  - Placa_175 [part] at (1150, 250, 200) mm
  - Disco_176 [part] at (1250, 230, 200) mm
  - Placa_177 [part] at (1150, 250, 200) mm
  - Disco_178 [part] at (1250, 230, 200) mm
  - Placa_179 [part] at (1146.4, 250, 200) mm
  - Placa_180 [part] at (1150, 250, 200) mm
  - Disco_181 [part] at (1250, 230, 200) mm
  - Placa_182 [part] at (1150, 250, 200) mm
  - Placa_183 [part] at (1150, 250, 200) mm
  - Placa_184 [part] at (1150, 250, 200) mm
  - Disco_185 [part] at (1250, 230, 200) mm
  - Placa_186 [part] at (1150, 250, 200) mm
  - Disco_187 [part] at (1250, 230, 200) mm
  - Disco_188 [part] at (1250, 230, 200) mm
  - Placa_189 [part] at (1150, 250, 200) mm
  - Placa_190 [part] at (1150, 250, 200) mm
  - Placa_191 [part] at (1150, 250, 200) mm
  - Placa_192 [part] at (1150, 250, 200) mm
  - Disco_193 [part] at (1250, 230, 200) mm
  - Placa_194 [part] at (1150, 250, 200) mm
  - Placa_195 [part] at (1150, 250, 200) mm
  - Disco_196 [part] at (1250, 230, 200) mm
  - Disco_197 [part] at (1250, 230, 200) mm
  - Placa_198 [part] at (1150, 250, 200) mm
  - Disco_199 [part] at (1250, 230, 200) mm
  - Disco_200 [part] at (1250, 230, 200) mm
  - Disco_201 [part] at (1250, 230, 200) mm
  - Placa_202 [part] at (1150, 250, 200) mm
  - Placa_203 [part] at (1146.4, 250, 200) mm
  - Disco_204 [part] at (1250, 230, 200) mm
  - Placa_205 [part] at (1150, 250, 200) mm
  - Disco_206 [part] at (1250, 230, 200) mm
  - Placa_207 [part] at (1150, 250, 200) mm
  - Placa_208 [part] at (1150, 250, 200) mm
  - Disco_209 [part] at (1250, 230, 200) mm
  - Disco_210 [part] at (1250, 230, 200) mm
  - Disco_211 [part] at (1246.4, 230, 200) mm
  - Placa_212 [part] at (1150, 250, 200) mm
  - Disco_213 [part] at (1250, 230, 200) mm
  - Placa_214 [part] at (1150, 250, 200) mm
  - Placa_215 [part] at (1150, 250, 200) mm
  - Placa_216 [part] at (1150, 250, 200) mm
  - Disco_217 [part] at (1250, 230, 200) mm
  - Placa_218 [part] at (1150, 250, 200) mm
  - Disco_219 [part] at (1250, 230, 200) mm
  - Disco_220 [part] at (1246.4, 230, 200) mm
  - Disco_221 [part] at (1250, 230, 200) mm
  - Disco_222 [part] at (1250, 230, 200) mm
  - Disco_223 [part] at (1250, 230, 200) mm
  - Disco_224 [part] at (1250, 230, 200) mm
  - Disco_225 [part] at (1250, 230, 200) mm
  - Placa_226 [part] at (1150, 250, 200) mm
  - Placa_227 [part] at (1150, 250, 200) mm
  - Disco_228 [part] at (1250, 230, 200) mm
  - Disco_229 [part] at (1250, 230, 200) mm
  - Placa_230 [part] at (1150, 250, 200) mm
  - Disco_231 [part] at (1250, 230, 200) mm
  - Placa_232 [part] at (1150, 250, 200) mm
  - Placa_233 [part] at (1150, 250, 200) mm
  - Placa_234 [part] at (1150, 250, 200) mm
  - Placa_235 [part] at (1150, 250, 200) mm
  - Disco_236 [part] at (1250, 230, 200) mm
  - Disco_237 [part] at (1250, 230, 200) mm
  - Placa_238 [part] at (1150, 250, 200) mm
  - Disco_239 [part] at (1250, 230, 200) mm
  - Disco_240 [part] at (1250, 230, 200) mm
  - Placa_241 [part] at (1150, 250, 200) mm
  - Placa_242 [part] at (1150, 250, 200) mm
  - Placa_243 [part] at (1150, 250, 200) mm
  - Disco_244 [part] at (1250, 230, 200) mm
  - Disco_245 [part] at (1246.4, 230, 200) mm
  - Disco_246 [part] at (1250, 230, 200) mm
  - Placa_247 [part] at (1150, 250, 200) mm
  - Disco_248 [part] at (1250, 230, 200) mm
  - Placa_249 [part] at (1150, 250, 200) mm
  - Placa_250 [part] at (1150, 250, 200) mm
  - Disco_251 [part] at (1250, 230, 200) mm
  - Placa_252 [part] at (1150, 250, 200) mm
  - Placa_253 [part] at (1146.4, 250, 200) mm
  - Placa_254 [part] at (1150, 250, 200) mm
  - Placa_255 [part] at (1150, 250, 200) mm
  - Placa_256 [part] at (1150, 250, 200) mm
  - Placa_257 [part] at (1150, 250, 200) mm
  - Disco_258 [part] at (1250, 230, 200) mm
  - Disco_259 [part] at (1250, 230, 200) mm
  - Placa_260 [part] at (1150, 250, 200) mm
  - Placa_261 [part] at (1146.4, 250, 200) mm
  - Placa_262 [part] at (1150, 250, 200) mm
  - Disco_263 [part] at (1250, 230, 200) mm
  - Placa_264 [part] at (1150, 250, 200) mm
  - Disco_265 [part] at (1250, 230, 200) mm
  - Placa_266 [part] at (1150, 250, 200) mm
  - Placa_267 [part] at (1150, 250, 200) mm
  - Disco_268 [part] at (1250, 230, 200) mm
  - Disco_269 [part] at (1250, 230, 200) mm
  - Placa_270 [part] at (1150, 250, 200) mm
  - Disco_271 [part] at (1250, 230, 200) mm
  - Disco_272 [part] at (1250, 230, 200) mm
  - Disco_273 [part] at (1250, 230, 200) mm
  - Disco_274 [part] at (1250, 230, 200) mm
  - Placa_275 [part] at (1150, 250, 200) mm
  - Placa_276 [part] at (1150, 250, 200) mm
  - Disco_277 [part] at (1250, 230, 200) mm
  - Placa_278 [part] at (1150, 250, 200) mm
  - Disco_279 [part] at (1250, 230, 200) mm
  - Disco_280 [part] at (1250, 230, 200) mm
  - Placa_281 [part] at (1150, 250, 200) mm
  - Disco_282 [part] at (1250, 230, 200) mm
  - Disco_283 [part] at (1250, 230, 200) mm
  - Disco_284 [part] at (1250, 230, 200) mm
  - Placa_285 [part] at (1146.4, 250, 200) mm
  - Disco_286 [part] at (1250, 230, 200) mm
  - Disco_287 [part] at (1250, 230, 200) mm
  - Disco_288 [part] at (1250, 230, 200) mm
  - Disco_289 [part] at (1250, 230, 200) mm
  - Placa_290 [part] at (1150, 250, 200) mm
  - Placa_291 [part] at (1150, 250, 200) mm
  - Placa_292 [part] at (1150, 250, 200) mm
  - Disco_293 [part] at (1246.4, 230, 200) mm
  - Placa_294 [part] at (1150, 250, 200) mm
  - Disco_295 [part] at (1250, 230, 200) mm
  - Disco_296 [part] at (1250, 230, 200) mm
  - Disco_297 [part] at (1250, 230, 200) mm
  - Disco_298 [part] at (1250, 230, 200) mm
  - Disco_299 [part] at (1250, 230, 200) mm
  - Disco_300 [part] at (1250, 230, 200) mm
  - Disco_301 [part] at (1250, 230, 200) mm
  - Disco_302 [part] at (1250, 230, 200) mm
  - Disco_303 [part] at (1250, 230, 200) mm
  - Disco_304 [part] at (1250, 230, 200) mm
  - Placa_305 [part] at (1150, 250, 200) mm
  - Placa_306 [part] at (1150, 250, 200) mm
  - Placa_307 [part] at (1150, 250, 200) mm
  - Disco_308 [part] at (1250, 230, 200) mm
  - Disco_309 [part] at (1246.4, 230, 200) mm
  - Disco_310 [part] at (1250, 230, 200) mm
  - Disco_311 [part] at (1250, 230, 200) mm
  - Placa_312 [part] at (1150, 250, 200) mm
  - Disco_313 [part] at (1250, 230, 200) mm
  - Disco_314 [part] at (1250, 230, 200) mm
  - Placa_315 [part] at (1150, 250, 200) mm
  - Placa_316 [part] at (1150, 250, 200) mm
  - Disco_317 [part] at (1250, 230, 200) mm
  - Disco_338 [part] at (1246.4, 230, 200) mm
  - Disco_355 [part] at (1250, 230, 200) mm
  - Placa_356 [part] at (1150, 250, 200) mm
  - Disco_357 [part] at (1250, 230, 200) mm
  - Disco_358 [part] at (1250, 230, 200) mm
  - Disco_359 [part] at (1250, 230, 200) mm
  - Disco_360 [part] at (1250, 230, 200) mm
  - Placa_361 [part] at (1150, 250, 200) mm
  - Disco_362 [part] at (1250, 230, 200) mm
  - Placa_363 [part] at (1150, 250, 200) mm
  - Disco_364 [part] at (1246.4, 230, 200) mm
  - Placa_365 [part] at (1150, 250, 200) mm
  - Disco_366 [part] at (1250, 230, 200) mm
  - Placa_367 [part] at (1150, 250, 200) mm
  - Placa_368 [part] at (1150, 250, 200) mm
  - Disco_369 [part] at (1250, 230, 200) mm
  - Disco_370 [part] at (1250, 230, 200) mm
  - Disco_371 [part] at (1250, 230, 200) mm
  - Placa_372 [part] at (1146.4, 250, 200) mm
  - Disco_373 [part] at (1250, 230, 200) mm
  - Disco_374 [part] at (1250, 230, 200) mm
  - Disco_375 [part] at (1250, 230, 200) mm
  - Disco_376 [part] at (1250, 230, 200) mm
  - Disco_377 [part] at (1250, 230, 200) mm
  - Disco_378 [part] at (1250, 230, 200) mm
  - Placa_379 [part] at (1150, 250, 200) mm
  - Placa_380 [part] at (1146.4, 250, 200) mm
  - Placa_381 [part] at (1150, 250, 200) mm
  - Placa_382 [part] at (1150, 250, 200) mm
  - Disco_383 [part] at (1250, 230, 200) mm
  - Placa_384 [part] at (1150, 250, 200) mm
  - Placa_385 [part] at (1150, 250, 200) mm
  - Placa_386 [part] at (1150, 250, 200) mm
  - Placa_387 [part] at (1150, 250, 200) mm
  - Placa_388 [part] at (1150, 250, 200) mm
  - Placa_389 [part] at (1150, 250, 200) mm
  - Disco_390 [part] at (1250, 230, 200) mm
  - Disco_391 [part] at (1250, 230, 200) mm
  - Placa_392 [part] at (1150, 250, 200) mm
  - Disco_393 [part] at (1250, 230, 200) mm
  - Disco_394 [part] at (1250, 230, 200) mm
  - Disco_395 [part] at (1250, 230, 200) mm
  - Disco_396 [part] at (1246.4, 230, 200) mm
  - Disco_397 [part] at (1250, 230, 200) mm
  - Placa_398 [part] at (1150, 250, 200) mm
  - Placa_399 [part] at (1150, 250, 200) mm
  - Disco_400 [part] at (1250, 230, 200) mm
  - Disco_401 [part] at (1250, 230, 200) mm
  - Disco_402 [part] at (1250, 230, 200) mm
  - Disco_403 [part] at (1250, 230, 200) mm
  - Disco_404 [part] at (1246.4, 230, 200) mm
  - Placa_405 [part] at (1150, 250, 200) mm
  - Placa_406 [part] at (1150, 250, 200) mm
  - Disco_407 [part] at (1250, 230, 200) mm
  - Disco_408 [part] at (1250, 230, 200) mm
  - Disco_409 [part] at (1250, 230, 200) mm
  - Placa_410 [part] at (1150, 250, 200) mm
  - Disco_411 [part] at (1250, 230, 200) mm
  - Disco_412 [part] at (1246.4, 230, 200) mm
  - Placa_413 [part] at (1150, 250, 200) mm
  - Placa_414 [part] at (1150, 250, 200) mm
  - Placa_415 [part] at (1150, 250, 200) mm
  - Placa_416 [part] at (1150, 250, 200) mm
  - Placa_417 [part] at (1150, 250, 200) mm
  - Placa_418 [part] at (1150, 250, 200) mm
  - Disco_419 [part] at (1250, 230, 200) mm
  - Placa_420 [part] at (1146.4, 250, 200) mm
  - Disco_421 [part] at (1250, 230, 200) mm
  - Placa_422 [part] at (1150, 250, 200) mm
  - Disco_423 [part] at (1250, 230, 200) mm
  - Disco_424 [part] at (1250, 230, 200) mm
  - Disco_425 [part] at (1250, 230, 200) mm
  - Disco_426 [part] at (1250, 230, 200) mm
  - Placa_427 [part] at (1150, 250, 200) mm
  - Placa_428 [part] at (1146.4, 250, 200) mm
  - Disco_429 [part] at (1250, 230, 200) mm
  - Disco_430 [part] at (1250, 230, 200) mm
  - Disco_431 [part] at (1250, 230, 200) mm
  - Disco_432 [part] at (1250, 230, 200) mm
  - Disco_433 [part] at (1250, 230, 200) mm
  - Placa_434 [part] at (1150, 250, 200) mm
  - Disco_435 [part] at (1250, 230, 200) mm
  - Placa_436 [part] at (1146.4, 250, 200) mm
  - Placa_437 [part] at (1150, 250, 200) mm
  - Disco_438 [part] at (1250, 230, 200) mm
  - Disco_439 [part] at (1250, 230, 200) mm
  - Disco_440 [part] at (1250, 230, 200) mm
  - Placa_441 [part] at (1150, 250, 200) mm
  - Disco_442 [part] at (1250, 230, 200) mm
  - Placa_443 [part] at (1150, 250, 200) mm
  - Placa_444 [part] at (1146.4, 250, 200) mm
  - Placa_445 [part] at (1150, 250, 200) mm
  - Disco_446 [part] at (1250, 230, 200) mm
  - Disco_447 [part] at (1250, 230, 200) mm
  - Placa_448 [part] at (1150, 250, 200) mm
  - Placa_449 [part] at (1150, 250, 200) mm
  - Disco_450 [part] at (1250, 230, 200) mm
  - Disco_451 [part] at (1250, 230, 200) mm
  - Disco_452 [part] at (1246.4, 230, 200) mm
  - Placa_453 [part] at (1150, 250, 200) mm
  - Disco_454 [part] at (1250, 230, 200) mm
  - Placa_455 [part] at (1150, 250, 200) mm
  - Disco_456 [part] at (1250, 230, 200) mm
  - Placa_457 [part] at (1150, 250, 200) mm
  - Placa_458 [part] at (1150, 250, 200) mm
  - Placa_459 [part] at (1150, 250, 200) mm
  - Disco_460 [part] at (1246.4, 230, 200) mm
  - Placa_461 [part] at (1150, 250, 200) mm
  - Placa_462 [part] at (1150, 250, 200) mm
  - Placa_463 [part] at (1150, 250, 200) mm
  - Placa_464 [part] at (1150, 250, 200) mm
  - Disco_465 [part] at (1250, 230, 200) mm
  - Placa_466 [part] at (1150, 250, 200) mm
  - Placa_467 [part] at (1150, 250, 200) mm
  - Disco_468 [part] at (1246.4, 230, 200) mm
  - Disco_469 [part] at (1250, 230, 200) mm
  - Disco_470 [part] at (1250, 230, 200) mm
  - Disco_471 [part] at (1250, 230, 200) mm
  - Placa_472 [part] at (1150, 250, 200) mm
  - Placa_473 [part] at (1150, 250, 200) mm
  - Placa_474 [part] at (1150, 250, 200) mm
  - Disco_475 [part] at (1250, 230, 200) mm
  - Disco_476 [part] at (1250, 230, 200) mm
  - Placa_477 [part] at (1150, 250, 200) mm
  - Disco_478 [part] at (1250, 230, 200) mm
  - Disco_479 [part] at (1250, 230, 200) mm
  - Disco_480 [part] at (1250, 230, 200) mm
  - Disco_481 [part] at (1250, 230, 200) mm
  - Placa_482 [part] at (1150, 250, 200) mm
  - Placa_483 [part] at (1150, 250, 200) mm
  - Disco_484 [part] at (1246.4, 230, 200) mm
  - Placa_485 [part] at (1150, 250, 200) mm
  - Disco_486 [part] at (1250, 230, 200) mm
  - Placa_487 [part] at (1150, 250, 200) mm
  - Disco_488 [part] at (1250, 230, 200) mm
  - Disco_489 [part] at (1250, 230, 200) mm
  - Placa_490 [part] at (1150, 250, 200) mm
  - Placa_491 [part] at (1150, 250, 200) mm
  - Placa_492 [part] at (1146.4, 250, 200) mm
  - Disco_493 [part] at (1250, 230, 200) mm
  - Disco_494 [part] at (1250, 230, 200) mm
  - Disco_495 [part] at (1250, 230, 200) mm
  - Placa_496 [part] at (1150, 250, 200) mm
  - Disco_497 [part] at (1250, 230, 200) mm
  - Placa_498 [part] at (1150, 250, 200) mm
  - Placa_499 [part] at (1150, 250, 200) mm
  - Placa_500 [part] at (1150, 250, 200) mm
  - Disco_501 [part] at (1250, 230, 200) mm
  - Disco_502 [part] at (1246.4, 230, 200) mm
  - Placa_505 [part] at (1146.4, 250, 200) mm
  - Placa_506 [part] at (1146.4, 250, 200) mm
  - Disco_18 [part] at (1250, 230, 200) mm
  - Disco_19 [part] at (1250, 230, 200) mm
  - Disco_20 [part] at (1250, 230, 200) mm
  - Placa_21 [part] at (1150, 250, 200) mm
  - Disco_22 [part] at (1250, 230, 200) mm
  - Disco_23 [part] at (1250, 230, 200) mm
  - Disco_24 [part] at (1250, 230, 200) mm
  - Placa_25 [part] at (1150, 250, 200) mm
  - Placa_26 [part] at (1150, 250, 200) mm
  - Placa_27 [part] at (1150, 250, 200) mm
  - Placa_28 [part] at (1150, 250, 200) mm
  - Disco_29 [part] at (1250, 230, 200) mm
  - Placa_30 [part] at (1150, 250, 200) mm
  - Placa_31 [part] at (1146.4, 250, 200) mm
  - Disco_32 [part] at (1250, 230, 200) mm
  - Placa_33 [part] at (1150, 250, 200) mm
  - Disco_34 [part] at (1250, 230, 200) mm
  - Disco_35 [part] at (1250, 230, 200) mm
  - Placa_36 [part] at (1150, 250, 200) mm
  - Disco_37 [part] at (1250, 230, 200) mm
  - Placa_38 [part] at (1146.4, 250, 200) mm
  - Placa_39 [part] at (1150, 250, 200) mm
  - Placa_40 [part] at (1146.4, 250, 200) mm
  - Placa_41 [part] at (1150, 250, 200) mm
  - Placa_42 [part] at (1146.4, 250, 200) mm
  - Disco_43 [part] at (1250, 230, 200) mm
  - Placa_44 [part] at (1146.4, 250, 200) mm
  - Placa_45 [part] at (1150, 250, 200) mm
  - Disco_46 [part] at (1250, 230, 200) mm
  - Disco_89 [part] at (1250, 230, 200) mm
  - Disco_90 [part] at (1250, 230, 200) mm
  - Disco_91 [part] at (1250, 230, 200) mm
  - Disco_92 [part] at (1246.4, 230, 200) mm
  - Placa_93 [part] at (1150, 250, 200) mm
  - Disco_94 [part] at (1250, 230, 200) mm
  - Placa_95 [part] at (1150, 250, 200) mm
  - Placa_96 [part] at (1150, 250, 200) mm
  - Disco_97 [part] at (1250, 230, 200) mm
  - Placa_98 [part] at (1150, 250, 200) mm
  - Placa_99 [part] at (1146.4, 250, 200) mm
  - Disco_100 [part] at (1250, 230, 200) mm
  - Disco_101 [part] at (1250, 230, 200) mm
  - Placa_102 [part] at (1150, 250, 200) mm
  - Placa_103 [part] at (1150, 250, 200) mm
  - Placa_104 [part] at (1150, 250, 200) mm
  - Placa_105 [part] at (1150, 250, 200) mm
  - Placa_106 [part] at (1146.4, 250, 200) mm
  - Placa_107 [part] at (1150, 250, 200) mm
  - Placa_108 [part] at (1150, 250, 200) mm
  - Placa_109 [part] at (1150, 250, 200) mm
  - Disco_110 [part] at (1250, 230, 200) mm
  - Placa_111 [part] at (1150, 250, 200) mm
  - Disco_112 [part] at (1250, 230, 200) mm
  - Disco_113 [part] at (1250, 230, 200) mm
  - Placa_114 [part] at (1150, 250, 200) mm
  - Disco_115 [part] at (1250, 230, 200) mm
  - Placa_116 [part] at (1150, 250, 200) mm
  - Placa_117 [part] at (1150, 250, 200) mm
  - Placa_118 [part] at (1150, 250, 200) mm
  - Disco_119 [part] at (1246.4, 230, 200) mm
  - Placa_120 [part] at (1150, 250, 200) mm
  - Placa_121 [part] at (1150, 250, 200) mm
  - Placa_122 [part] at (1150, 250, 200) mm
  - Disco_123 [part] at (1250, 230, 200) mm
  - Placa_124 [part] at (1150, 250, 200) mm
  - Placa_125 [part] at (1150, 250, 200) mm
  - Disco_126 [part] at (1246.4, 230, 200) mm
  - Placa_127 [part] at (1150, 250, 200) mm
  - Disco_128 [part] at (1250, 230, 200) mm
  - Disco_129 [part] at (1250, 230, 200) mm
  - Placa_130 [part] at (1150, 250, 200) mm
  - Placa_131 [part] at (1150, 250, 200) mm
  - Placa_132 [part] at (1150, 250, 200) mm
  - Disco_133 [part] at (1246.4, 230, 200) mm
  - Disco_134 [part] at (1250, 230, 200) mm
  - Disco_135 [part] at (1250, 230, 200) mm
  - Disco_136 [part] at (1250, 230, 200) mm
  - Disco_137 [part] at (1250, 230, 200) mm
  - Placa_138 [part] at (1150, 250, 200) mm
  - Disco_139 [part] at (1250, 230, 200) mm
  - Disco_140 [part] at (1250, 230, 200) mm
  - Placa_23 [part] at (1146.4, 250, 200) mm
  - Disco_38 [part] at (1246.4, 230, 200) mm
  - Placa_39 [part] at (1146.4, 250, 200) mm
  - Placa_40 [part] at (1150, 250, 200) mm
  - Placa_41 [part] at (1150, 250, 200) mm
  - Placa_42 [part] at (1150, 250, 200) mm
  - Disco_43 [part] at (1250, 230, 200) mm
  - Disco_44 [part] at (1250, 230, 200) mm
  - Placa_45 [part] at (1150, 250, 200) mm
  - Placa_46 [part] at (1146.4, 250, 200) mm
  - Disco_47 [part] at (1250, 230, 200) mm
  - Disco_48 [part] at (1250, 230, 200) mm
  - Disco_49 [part] at (1250, 230, 200) mm
  - Disco_50 [part] at (1250, 230, 200) mm
  - Placa_51 [part] at (1150, 250, 200) mm
  - Placa_52 [part] at (1150, 250, 200) mm
  - Placa_53 [part] at (1150, 250, 200) mm
  - Disco_54 [part] at (1250, 230, 200) mm
  - Placa_55 [part] at (1150, 250, 200) mm
  - Placa_56 [part] at (1150, 250, 200) mm
  - Placa_57 [part] at (1150, 250, 200) mm
  - Disco_58 [part] at (1250, 230, 200) mm
  - Disco_59 [part] at (1250, 230, 200) mm
  - Placa_60 [part] at (1146.4, 250, 200) mm
  - Placa_61 [part] at (1150, 250, 200) mm
  - Disco_62 [part] at (1250, 230, 200) mm
  - Placa_63 [part] at (1150, 250, 200) mm
  - Placa_64 [part] at (1150, 250, 200) mm
  - Disco_65 [part] at (1250, 230, 200) mm
  - Disco_66 [part] at (1250, 230, 200) mm
  - Disco_67 [part] at (1246.4, 230, 200) mm
  - Disco_68 [part] at (1250, 230, 200) mm
  - Disco_69 [part] at (1250, 230, 200) mm
  - Placa_70 [part] at (1150, 250, 200) mm
  - Placa_71 [part] at (1150, 250, 200) mm
  - Disco_72 [part] at (1250, 230, 200) mm
  - Disco_73 [part] at (1250, 230, 200) mm
  - Disco_74 [part] at (1246.4, 230, 200) mm
  - Disco_75 [part] at (1250, 230, 200) mm
  - Disco_76 [part] at (1250, 230, 200) mm
  - Disco_77 [part] at (1250, 230, 200) mm
  - Disco_78 [part] at (1250, 230, 200) mm
  - Disco_79 [part] at (1250, 230, 200) mm
  - Disco_80 [part] at (1250, 230, 200) mm
  - Placa_81 [part] at (1146.4, 250, 200) mm
  - Disco_82 [part] at (1250, 230, 200) mm
  - Disco_83 [part] at (1250, 230, 200) mm
  - Placa_84 [part] at (1150, 250, 200) mm
  - Disco_85 [part] at (1250, 230, 200) mm
  - Placa_86 [part] at (1150, 250, 200) mm
  - Placa_87 [part] at (1150, 250, 200) mm
  - Placa_88 [part] at (1146.4, 250, 200) mm
  - Placa_89 [part] at (1150, 250, 200) mm
  - Placa_90 [part] at (1150, 250, 200) mm
  - Disco_91 [part] at (1250, 230, 200) mm
  - Placa_92 [part] at (1150, 250, 200) mm
  - Placa_93 [part] at (1150, 250, 200) mm
  - Placa_94 [part] at (1150, 250, 200) mm
  - Placa_95 [part] at (1146.4, 250, 200) mm
  - Disco_96 [part] at (1250, 230, 200) mm
  - Placa_97 [part] at (1150, 250, 200) mm
  - Placa_98 [part] at (1150, 250, 200) mm
  - Disco_99 [part] at (1250, 230, 200) mm
  - Placa_100 [part] at (1150, 250, 200) mm
  - Disco_101 [part] at (1250, 230, 200) mm
  - Placa_102 [part] at (1146.4, 250, 200) mm
  - Disco_103 [part] at (1250, 230, 200) mm
  - Disco_104 [part] at (1250, 230, 200) mm
  - Placa_105 [part] at (1150, 250, 200) mm
  - Placa_106 [part] at (1150, 250, 200) mm
  - Placa_107 [part] at (1150, 250, 200) mm
  - Placa_108 [part] at (1150, 250, 200) mm
  - Placa_109 [part] at (1146.4, 250, 200) mm
  - Disco_110 [part] at (1250, 230, 200) mm
  - Disco_111 [part] at (1250, 230, 200) mm
  - Disco_112 [part] at (1250, 230, 200) mm
  - Placa_113 [part] at (1150, 250, 200) mm
  - Disco_114 [part] at (1250, 230, 200) mm
  - Disco_115 [part] at (1250, 230, 200) mm
  - Placa_116 [part] at (1146.4, 250, 200) mm
  - Placa_117 [part] at (1150, 250, 200) mm
  - Placa_118 [part] at (1150, 250, 200) mm
  - Placa_119 [part] at (1150, 250, 200) mm
  - Disco_120 [part] at (1250, 230, 200) mm
  - Placa_121 [part] at (1150, 250, 200) mm
  - Placa_122 [part] at (1150, 250, 200) mm
  - Placa_123 [part] at (1146.4, 250, 200) mm
  - Disco_124 [part] at (1250, 230, 200) mm
  - Placa_125 [part] at (1150, 250, 200) mm
  - Placa_126 [part] at (1150, 250, 200) mm
  - Placa_127 [part] at (1150, 250, 200) mm
  - Disco_128 [part] at (1250, 230, 200) mm
  - Disco_129 [part] at (1250, 230, 200) mm
  - Disco_130 [part] at (1246.4, 230, 200) mm
  - Placa_131 [part] at (1150, 250, 200) mm
  - Placa_132 [part] at (1150, 250, 200) mm
  - Placa_133 [part] at (1150, 250, 200) mm
  - Placa_134 [part] at (1150, 250, 200) mm
  - Placa_135 [part] at (1150, 250, 200) mm
  - Placa_136 [part] at (1150, 250, 200) mm
  - Placa_137 [part] at (1146.4, 250, 200) mm
  - Placa_138 [part] at (1150, 250, 200) mm
  - Disco_139 [part] at (1250, 230, 200) mm
  - Disco_140 [part] at (1250, 230, 200) mm
  - Disco_141 [part] at (1250, 230, 200) mm
  - Placa_142 [part] at (1150, 250, 200) mm
  - Placa_143 [part] at (1150, 250, 200) mm
  - Disco_144 [part] at (1246.4, 230, 200) mm
  - Disco_145 [part] at (1250, 230, 200) mm
  - Placa_146 [part] at (1150, 250, 200) mm
  - Disco_147 [part] at (1250, 230, 200) mm
  - Disco_148 [part] at (1250, 230, 200) mm
  - Disco_149 [part] at (1250, 230, 200) mm
  - Disco_150 [part] at (1250, 230, 200) mm
  - Disco_151 [part] at (1246.4, 230, 200) mm
  - Disco_152 [part] at (1250, 230, 200) mm
  - Placa_153 [part] at (1150, 250, 200) mm
  - Disco_154 [part] at (1250, 230, 200) mm
  - Placa_155 [part] at (1150, 250, 200) mm
  - Disco_156 [part] at (1250, 230, 200) mm
  - Placa_157 [part] at (1150, 250, 200) mm
  - Placa_158 [part] at (1150, 250, 200) mm
  - Placa_159 [part] at (1150, 250, 200) mm
  - Disco_160 [part] at (1250, 230, 200) mm
  - Disco_161 [part] at (1250, 230, 200) mm
  - Disco_162 [part] at (1250, 230, 200) mm
  - Placa_163 [part] at (1150, 250, 200) mm
  - Placa_164 [part] at (1150, 250, 200) mm
  - Placa_165 [part] at (1146.4, 250, 200) mm
  - Placa_166 [part] at (1150, 250, 200) mm
  - Disco_167 [part] at (1250, 230, 200) mm
  - Placa_168 [part] at (1150, 250, 200) mm
  - Disco_169 [part] at (1250, 230, 200) mm
  - Placa_170 [part] at (1150, 250, 200) mm
  - Placa_171 [part] at (1150, 250, 200) mm
  - Placa_172 [part] at (1146.4, 250, 200) mm
  - Disco_173 [part] at (1250, 230, 200) mm
  - Disco_174 [part] at (1250, 230, 200) mm
  - Disco_175 [part] at (1250, 230, 200) mm
  - Placa_176 [part] at (1150, 250, 200) mm
  - Disco_177 [part] at (1250, 230, 200) mm
  - Placa_178 [part] at (1150, 250, 200) mm
  - Disco_179 [part] at (1246.4, 230, 200) mm
  - Placa_180 [part] at (1150, 250, 200) mm
  - Disco_181 [part] at (1250, 230, 200) mm
  - Disco_182 [part] at (1250, 230, 200) mm
  - Disco_183 [part] at (1250, 230, 200) mm
  - Placa_184 [part] at (1150, 250, 200) mm
  - Placa_185 [part] at (1150, 250, 200) mm
  - Disco_186 [part] at (1246.4, 230, 200) mm
  - Disco_187 [part] at (1250, 230, 200) mm
  - Placa_188 [part] at (1150, 250, 200) mm
  - Placa_189 [part] at (1150, 250, 200) mm
  - Disco_190 [part] at (1250, 230, 200) mm
  - Placa_191 [part] at (1150, 250, 200) mm
  - Placa_192 [part] at (1150, 250, 200) mm
  - Disco_193 [part] at (1246.4, 230, 200) mm
  - Disco_194 [part] at (1250, 230, 200) mm
  - Disco_195 [part] at (1250, 230, 200) mm
  - Disco_196 [part] at (1250, 230, 200) mm
  - Disco_197 [part] at (1250, 230, 200) mm
  - Placa_198 [part] at (1150, 250, 200) mm
  - Placa_199 [part] at (1150, 250, 200) mm
  - Placa_200 [part] at (1146.4, 250, 200) mm
  - Disco_201 [part] at (1250, 230, 200) mm
  - Disco_202 [part] at (1250, 230, 200) mm
  - Disco_203 [part] at (1250, 230, 200) mm
  - Placa_204 [part] at (1150, 250, 200) mm
  - Disco_205 [part] at (1250, 230, 200) mm
  - Disco_206 [part] at (1250, 230, 200) mm
  - Placa_207 [part] at (1146.4, 250, 200) mm
  - Disco_208 [part] at (1250, 230, 200) mm
  - Disco_209 [part] at (1250, 230, 200) mm
  - Placa_210 [part] at (1150, 250, 200) mm
  - Disco_211 [part] at (1250, 230, 200) mm
  - Disco_212 [part] at (1250, 230, 200) mm
  - Placa_213 [part] at (1150, 250, 200) mm
  - Placa_214 [part] at (1146.4, 250, 200) mm
  - Placa_215 [part] at (1150, 250, 200) mm
  - Disco_216 [part] at (1250, 230, 200) mm
  - Disco_217 [part] at (1250, 230, 200) mm
  - Placa_218 [part] at (1150, 250, 200) mm
  - Placa_219 [part] at (1150, 250, 200) mm
  - Disco_220 [part] at (1250, 230, 200) mm
  - Placa_221 [part] at (1146.4, 250, 200) mm
  - Placa_222 [part] at (1150, 250, 200) mm
  - Placa_223 [part] at (1150, 250, 200) mm
  - Placa_224 [part] at (1150, 250, 200) mm
  - Placa_225 [part] at (1150, 250, 200) mm
  - Disco_226 [part] at (1250, 230, 200) mm
  - Placa_227 [part] at (1150, 250, 200) mm
  - Disco_228 [part] at (1246.4, 230, 200) mm
  - Disco_229 [part] at (1250, 230, 200) mm
  - Disco_230 [part] at (1250, 230, 200) mm
  - Placa_231 [part] at (1150, 250, 200) mm
  - Disco_232 [part] at (1250, 230, 200) mm
  - Placa_233 [part] at (1150, 250, 200) mm
  - Disco_234 [part] at (1250, 230, 200) mm
  - Disco_235 [part] at (1246.4, 230, 200) mm
  - Placa_236 [part] at (1150, 250, 200) mm
  - Placa_237 [part] at (1150, 250, 200) mm
  - Disco_238 [part] at (1250, 230, 200) mm
  - Placa_239 [part] at (1150, 250, 200) mm
  - Placa_240 [part] at (1150, 250, 200) mm
  - Placa_241 [part] at (1150, 250, 200) mm
  - Placa_242 [part] at (1146.4, 250, 200) mm
  - Placa_243 [part] at (1150, 250, 200) mm
  - Disco_244 [part] at (1250, 230, 200) mm
  - Disco_245 [part] at (1250, 230, 200) mm
  - Disco_246 [part] at (1250, 230, 200) mm
  - Placa_247 [part] at (1150, 250, 200) mm
  - Disco_248 [part] at (1250, 230, 200) mm
  - Disco_249 [part] at (1246.4, 230, 200) mm
  - Disco_250 [part] at (1250, 230, 200) mm
  - Placa_251 [part] at (1150, 250, 200) mm
  - Placa_252 [part] at (1150, 250, 200) mm
  - Disco_253 [part] at (1250, 230, 200) mm
  - Placa_254 [part] at (1150, 250, 200) mm
  - Disco_255 [part] at (1250, 230, 200) mm
  - Placa_256 [part] at (1146.4, 250, 200) mm
  - Disco_257 [part] at (1250, 230, 200) mm
  - Disco_258 [part] at (1250, 230, 200) mm
  - Placa_259 [part] at (1150, 250, 200) mm
  - Disco_260 [part] at (1250, 230, 200) mm
  - Placa_261 [part] at (1150, 250, 200) mm
  - Disco_262 [part] at (1250, 230, 200) mm
  - Disco_263 [part] at (1246.4, 230, 200) mm
  - Disco_264 [part] at (1250, 230, 200) mm
  - Disco_265 [part] at (1250, 230, 200) mm
  - Disco_266 [part] at (1250, 230, 200) mm
  - Placa_267 [part] at (1150, 250, 200) mm
  - Placa_268 [part] at (1150, 250, 200) mm
  - Disco_269 [part] at (1250, 230, 200) mm
  - Placa_270 [part] at (1146.4, 250, 200) mm
  - Disco_271 [part] at (1250, 230, 200) mm
  - Placa_272 [part] at (1150, 250, 200) mm
  - Placa_273 [part] at (1150, 250, 200) mm
  - Disco_274 [part] at (1250, 230, 200) mm
  - Placa_275 [part] at (1150, 250, 200) mm
  - Placa_276 [part] at (1150, 250, 200) mm
  - Placa_277 [part] at (1146.4, 250, 200) mm
  - Placa_278 [part] at (1150, 250, 200) mm
  - Placa_279 [part] at (1150, 250, 200) mm
  - Disco_280 [part] at (1250, 230, 200) mm
  - Disco_281 [part] at (1250, 230, 200) mm
  - Disco_282 [part] at (1250, 230, 200) mm
  - Placa_283 [part] at (1150, 250, 200) mm
  - Placa_284 [part] at (1146.4, 250, 200) mm
  - Disco_285 [part] at (1250, 230, 200) mm
  - Disco_286 [part] at (1250, 230, 200) mm
  - Placa_287 [part] at (1150, 250, 200) mm
  - Disco_288 [part] at (1250, 230, 200) mm
  - Disco_289 [part] at (1250, 230, 200) mm
  - Placa_290 [part] at (1150, 250, 200) mm
  - Disco_291 [part] at (1246.4, 230, 200) mm
  - Placa_292 [part] at (1150, 250, 200) mm
  - Disco_293 [part] at (1250, 230, 200) mm
  - Placa_294 [part] at (1150, 250, 200) mm
  - Disco_295 [part] at (1250, 230, 200) mm
  - Disco_296 [part] at (1250, 230, 200) mm
  - Placa_297 [part] at (1150, 250, 200) mm
  - Placa_298 [part] at (1146.4, 250, 200) mm
  - Placa_299 [part] at (1150, 250, 200) mm
  - Placa_300 [part] at (1150, 250, 200) mm
  - Placa_301 [part] at (1150, 250, 200) mm
  - Disco_302 [part] at (1250, 230, 200) mm
  - Disco_303 [part] at (1250, 230, 200) mm
  - Disco_304 [part] at (1250, 230, 200) mm
  - Disco_305 [part] at (1246.4, 230, 200) mm
  - Disco_306 [part] at (1250, 230, 200) mm
  - Placa_307 [part] at (1150, 250, 200) mm
  - Placa_308 [part] at (1150, 250, 200) mm
  - Placa_309 [part] at (1150, 250, 200) mm
  - Placa_310 [part] at (1150, 250, 200) mm
  - Placa_311 [part] at (1150, 250, 200) mm
  - Placa_312 [part] at (1150, 250, 200) mm
  - Disco_313 [part] at (1250, 230, 200) mm
  - Placa_314 [part] at (1150, 250, 200) mm
  - Placa_315 [part] at (1150, 250, 200) mm
  - Disco_316 [part] at (1250, 230, 200) mm
  - Placa_317 [part] at (1150, 250, 200) mm
  - Disco_318 [part] at (1250, 230, 200) mm
  - Disco_358 [part] at (1250, 230, 200) mm
  - Placa_359 [part] at (1146.4, 250, 200) mm
  - Placa_360 [part] at (1146.4, 250, 200) mm
  - Placa_361 [part] at (1150, 250, 200) mm
  - Disco_362 [part] at (1250, 230, 200) mm
  - Placa_363 [part] at (1150, 250, 200) mm
  - Disco_364 [part] at (1250, 230, 200) mm
  - Placa_365 [part] at (1150, 250, 200) mm
  - Disco_366 [part] at (1250, 230, 200) mm
  - Placa_367 [part] at (1146.4, 250, 200) mm
  - Disco_368 [part] at (1250, 230, 200) mm
  - Disco_369 [part] at (1250, 230, 200) mm
  - Placa_370 [part] at (1150, 250, 200) mm
  - Disco_371 [part] at (1250, 230, 200) mm
  - Disco_372 [part] at (1250, 230, 200) mm
  - Disco_373 [part] at (1250, 230, 200) mm
  - Placa_374 [part] at (1146.4, 250, 200) mm
  - Disco_375 [part] at (1250, 230, 200) mm
  - Disco_376 [part] at (1250, 230, 200) mm
  - Disco_377 [part] at (1250, 230, 200) mm
  - Disco_378 [part] at (1250, 230, 200) mm
  - Placa_379 [part] at (1150, 250, 200) mm
  - Placa_380 [part] at (1150, 250, 200) mm
  - Placa_381 [part] at (1146.4, 250, 200) mm
  - Disco_382 [part] at (1250, 230, 200) mm
  - Disco_383 [part] at (1250, 230, 200) mm
  - Placa_384 [part] at (1150, 250, 200) mm
  - Placa_385 [part] at (1150, 250, 200) mm
  - Disco_386 [part] at (1250, 230, 200) mm
  - Placa_387 [part] at (1150, 250, 200) mm
  - Placa_388 [part] at (1146.4, 250, 200) mm
  - Placa_389 [part] at (1150, 250, 200) mm
  - Disco_390 [part] at (1250, 230, 200) mm
  - Disco_391 [part] at (1250, 230, 200) mm
  - Placa_392 [part] at (1150, 250, 200) mm
  - Placa_393 [part] at (1150, 250, 200) mm
  - Placa_394 [part] at (1150, 250, 200) mm
  - Disco_395 [part] at (1246.4, 230, 200) mm
  - Disco_396 [part] at (1250, 230, 200) mm
  - Disco_397 [part] at (1250, 230, 200) mm
  - Placa_398 [part] at (1150, 250, 200) mm
  - Placa_399 [part] at (1150, 250, 200) mm
  - Placa_400 [part] at (1150, 250, 200) mm
  - Disco_401 [part] at (1250, 230, 200) mm
  - Disco_402 [part] at (1250, 230, 200) mm
  - Disco_14 [part] at (1246.4, 230, 200) mm
  - Disco_56 [part] at (1250, 230, 200) mm
  - Placa_57 [part] at (1146.4, 250, 200) mm
  - Disco_58 [part] at (1250, 230, 200) mm
  - Placa_59 [part] at (1150, 250, 200) mm
  - Disco_60 [part] at (1250, 230, 200) mm
  - Placa_61 [part] at (1150, 250, 200) mm
  - Placa_62 [part] at (1150, 250, 200) mm
  - Placa_63 [part] at (1150, 250, 200) mm
  - Placa_64 [part] at (1150, 250, 200) mm
  - Disco_79 [part] at (467.49, -181.23, 169.29) mm, rotated rx -0.77 ry -3.42 rz 6.56 deg
  - Placa_80 [part] at (476.98, -221.26, 8.17) mm, rotated rx -0.32 ry -2.05 rz -0.53 deg
  - Placa_81 [part] at (476.98, -221.26, 48.17) mm, rotated rx -0.32 ry -2.05 rz -0.53 deg
  - Placa_82 [part] at (336.98, -221.23, 8.25) mm, rotated rx -0.32 ry -2.05 rz -0.53 deg
  - Disco_83 [part] at (-30.88, -444.88, 157.75) mm, rotated rx 0.03 ry -1.07 rz 133.39 deg
  - Placa_84 [part] at (336.98, -221.25, 48.19) mm, rotated rx -0.32 ry -2.05 rz -0.53 deg
  - Placa_85 [part] at (31.62, -465.26, 122) mm, rotated rx -46.61 ry 88.76 rz 79.06 deg
  - Placa_86 [part] at (-3.38, -417.26, 122) mm, rotated rx -46.61 ry 88.76 rz 79.06 deg
  - Disco_87 [part] at (397.49, -181.23, 89.28) mm, rotated rx -0.77 ry -3.42 rz 6.56 deg
  - Placa_88 [part] at (37.45, -469.29, 118.84) mm, rotated rx 0.19 ry 0.39 rz 126.33 deg
  - Disco_89 [part] at (537.49, -181.23, 89.28) mm, rotated rx -0.77 ry -3.42 rz 6.56 deg
  - Placa_90 [part] at (406.97, -221.24, 128.2) mm, rotated rx -0.32 ry -2.05 rz -0.53 deg
  - Placa_91 [part] at (149.2, 250, 200) mm
  - Disco_92 [part] at (1246.4, 230, 200) mm
  - Placa_93 [part] at (1146.4, 250, 200) mm
  - Disco_94 [part] at (1246.4, 230, 200) mm
  - Disco_95 [part] at (1250, 230, 200) mm
  - Disco_96 [part] at (1250, 230, 200) mm
  - Placa_97 [part] at (1150, 250, 200) mm
  - Disco_98 [part] at (1250, 230, 200) mm
  - Disco_99 [part] at (1250, 230, 200) mm
  - Placa_100 [part] at (1150, 250, 200) mm
  - Disco_101 [part] at (1246.4, 230, 200) mm
  - Placa_102 [part] at (1150, 250, 200) mm
  - Placa_103 [part] at (1150, 250, 200) mm
  - Disco_104 [part] at (1250, 230, 200) mm
  - Disco_105 [part] at (1250, 230, 200) mm
  - Placa_106 [part] at (1150, 250, 200) mm
  - Disco_107 [part] at (1250, 230, 200) mm
  - Placa_108 [part] at (1146.4, 250, 200) mm
  - Disco_109 [part] at (1250, 230, 200) mm
  - Placa_110 [part] at (1150, 250, 200) mm
  - Placa_111 [part] at (1150, 250, 200) mm
  - Disco_112 [part] at (1250, 230, 200) mm
  - Disco_113 [part] at (1250, 230, 200) mm
  - Disco_114 [part] at (1250, 230, 200) mm
  - Placa_115 [part] at (1146.4, 250, 200) mm
  - Disco_116 [part] at (1250, 230, 200) mm
  - Placa_117 [part] at (1150, 250, 200) mm
  - Disco_118 [part] at (1250, 230, 200) mm
  - Disco_119 [part] at (1250, 230, 200) mm
  - Disco_120 [part] at (1250, 230, 200) mm
  - Disco_121 [part] at (1250, 230, 200) mm
  - Disco_122 [part] at (1246.4, 230, 200) mm
  - Disco_123 [part] at (1250, 230, 200) mm
  - Disco_124 [part] at (1250, 230, 200) mm
  - Placa_125 [part] at (1150, 250, 200) mm
  - Placa_126 [part] at (1150, 250, 200) mm
  - Disco_127 [part] at (1250, 230, 200) mm
  - Disco_128 [part] at (1250, 230, 200) mm
  - Placa_129 [part] at (1146.4, 250, 200) mm
  - Placa_130 [part] at (1150, 250, 200) mm
  - Disco_131 [part] at (1250, 230, 200) mm
  - Disco_132 [part] at (1250, 230, 200) mm
  - Placa_133 [part] at (1150, 250, 200) mm
  - Disco_134 [part] at (1250, 230, 200) mm
  - Placa_135 [part] at (1150, 250, 200) mm
  - Placa_136 [part] at (1146.4, 250, 200) mm
  - Placa_137 [part] at (1150, 250, 200) mm
  - Placa_138 [part] at (1150, 250, 200) mm
  - Disco_139 [part] at (1250, 230, 200) mm
  - Placa_140 [part] at (1150, 250, 200) mm
  - Disco_141 [part] at (1250, 230, 200) mm
  - Disco_142 [part] at (1250, 230, 200) mm
  - Placa_143 [part] at (1146.4, 250, 200) mm
  - Placa_144 [part] at (1150, 250, 200) mm
  - Disco_145 [part] at (1250, 230, 200) mm
  - Disco_146 [part] at (1250, 230, 200) mm
  - Disco_147 [part] at (1250, 230, 200) mm
  - Disco_148 [part] at (1250, 230, 200) mm
  - Disco_149 [part] at (1250, 230, 200) mm
  - Disco_150 [part] at (1246.4, 230, 200) mm
  - Disco_151 [part] at (1250, 230, 200) mm
  - Disco_152 [part] at (1250, 230, 200) mm
  - Placa_153 [part] at (1150, 250, 200) mm
  - Disco_154 [part] at (1250, 230, 200) mm
  - Placa_155 [part] at (1150, 250, 200) mm
  - Disco_156 [part] at (1250, 230, 200) mm
  - Placa_157 [part] at (1146.4, 250, 200) mm
  - Placa_158 [part] at (1150, 250, 200) mm
  - Disco_159 [part] at (1250, 230, 200) mm
  - Placa_160 [part] at (1150, 250, 200) mm
  - Disco_161 [part] at (1250, 230, 200) mm
  - Placa_162 [part] at (1150, 250, 200) mm
  - Placa_163 [part] at (1150, 250, 200) mm
  - Placa_164 [part] at (1146.4, 250, 200) mm
  - Disco_165 [part] at (1250, 230, 200) mm
  - Placa_166 [part] at (1150, 250, 200) mm
  - Placa_167 [part] at (1150, 250, 200) mm
  - Placa_168 [part] at (1150, 250, 200) mm
  - Placa_169 [part] at (1150, 250, 200) mm
  - Placa_170 [part] at (1150, 250, 200) mm
  - Disco_171 [part] at (1250, 230, 200) mm
Attachment: LineSensor is attached to MyNewTool / Cono
Attachment: MyNewTool is attached to IRB120_3_58__01 / Link6
Station logic (signal -> signal, property => property):
  CI_Cinta.SensorCinta1 -> CI_Piezas.Desencolar
  CI_Ventosa.Vacuostato -> IRB_120_3kg_0.58m_1.Vacuostato
  CI_Cinta.SensorCinta2 -> IRB_120_3kg_0.58m_1.SensorCinta2
  CI_Cinta.SensorCinta1 -> IRB_120_3kg_0.58m_1.SensorCinta1
  IRB_120_3kg_0.58m_1.Pieza -> CI_Piezas.Pieza
  IRB_120_3kg_0.58m_1.MotorCinta -> CI_Piezas.MotorCinta
  IRB_120_3kg_0.58m_1.ActivaVentosa -> CI_Ventosa.ActivaVentosa
  IRB_120_3kg_0.58m_1.ActivaSensores -> CI_Cinta.ActivaSensores

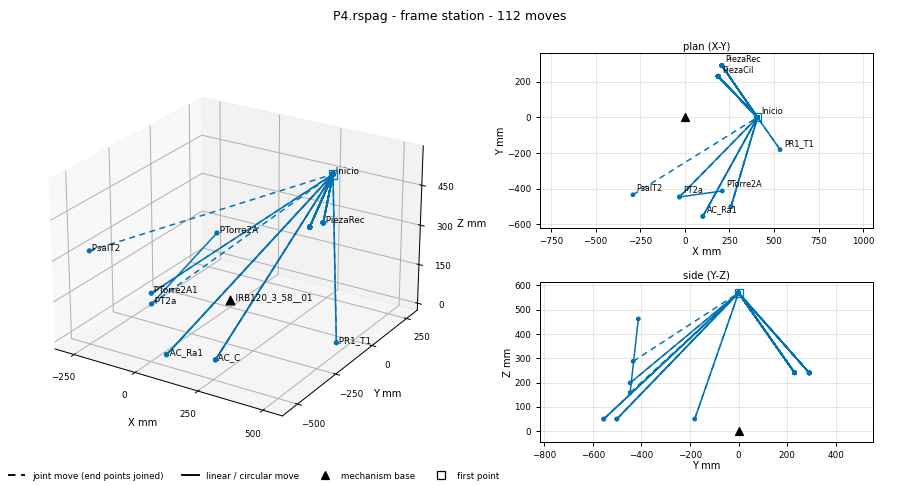
[picture p0: tool path of P4.rspag in frame station, 112 of 140 moves have a stored position in this frame; points joined in program order, loops and branches not executed]
--- Backups/IRB_120_3kg_0.58m_1/RAPID/TASK1/PROGMOD/CalibData.mod ---
MODULE CalibData
	PERS tooldata MyNewTool:=[TRUE,[[0,0,50],[1,0,0,0]],[1,[0,0,1],[1,0,0,0],0,0,0]];
ENDMODULE

--- Backups/IRB_120_3kg_0.58m_1/RAPID/TASK1/PROGMOD/Module1.mod ---
MODULE Module1
	CONST robtarget Target_10:=[[407.655094737,0,568.999992163],[0.499999968,0,0.866025422,0],[0,0,0,0],[9E+09,9E+09,9E+09,9E+09,9E+09,9E+09]];
    CONST robtarget Target_20:=[[189.2,230,240],[0,0,1,0],[0,0,0,0],[9E+09,9E+09,9E+09,9E+09,9E+09,9E+09]];
    CONST robtarget Inicio:=[[407.655094737,0,568.999992163],[0.499999968,0,0.866025422,0],[0,0,0,0],[9E+09,9E+09,9E+09,9E+09,9E+09,9E+09]];
    CONST robtarget PiezaRec:=[[207.655101241,291.000014691,239.998658793],[0.00319382,-0.090493869,0.995890978,-0.001348464],[0,-1,0,0],[9E+09,9E+09,9E+09,9E+09,9E+09,9E+09]];
    CONST robtarget PR1_T1:=[[534.35350098,-180.567604122,50.000737408],[0.020689968,-0.085804702,0.996080195,-0.00580719],[-1,0,-1,0],[9E+09,9E+09,9E+09,9E+09,9E+09,9E+09]];
    CONST robtarget AC_R:=[[32.752977258,-563.085746424,50.00068801],[0.013905422,0.485865655,0.873769287,-0.016384062],[-1,0,-1,0],[9E+09,9E+09,9E+09,9E+09,9E+09,9E+09]];
    CONST robtarget AC_C:=[[258.948994302,-501.082619671,50.000680143],[0.017008014,0.293581415,0.955692499,-0.013134953],[-1,0,-1,0],[9E+09,9E+09,9E+09,9E+09,9E+09,9E+09]];
    CONST robtarget PiezaCil:=[[187.395202706,230.469486387,240.836149731],[0.009317943,0.028928409,-0.999537888,-0.000578253],[0,0,0,0],[9E+09,9E+09,9E+09,9E+09,9E+09,9E+09]];
    VAR num aux:=1;
    VAR num estadoC:=1;
    VAR num estadoR:=1;
    VAR num listo:=0;
    VAR num estadoF:=1;

    CONST robtarget PR1_T2:=[[-462.931577079,-328.465147609,111.51088692],[0.676722375,0.713550687,0.03922699,0.177069162],[-2,1,-1,0],[9E+09,9E+09,9E+09,9E+09,9E+09,9E+09]];
    CONST robtarget PR1_T2a:=[[-532.244933646,-186.691334235,50.00073741],[0.001245183,0.91387717,0.405421658,-0.021453386],[-2,0,-1,0],[9E+09,9E+09,9E+09,9E+09,9E+09,9E+09]];
    CONST robtarget AC_C2:=[[372.479975366,-423.552888706,50.00068045],[0.01848201,0.174923473,0.984347488,-0.010964311],[-1,0,-1,0],[9E+09,9E+09,9E+09,9E+09,9E+09,9E+09]];

    CONST robtarget PR1_T2s:=[[-324.772773009,-455.442627096,63.510389948],[0.368990652,0.660928034,-0.271785572,0.594266468],[-2,1,0,0],[9E+09,9E+09,9E+09,9E+09,9E+09,9E+09]];
    CONST robtarget PR2_T2s:=[[-359.772705928,-407.442815025,63.510131305],[0.368990636,0.66092811,-0.271785282,0.594266526],[-2,0,0,0],[9E+09,9E+09,9E+09,9E+09,9E+09,9E+09]];
    CONST robtarget PR2_T2a:=[[-341.393194601,-446.15939263,164.008267513],[0.024998806,-0.922581412,0.38494258,-0.006148755],[-2,-1,1,0],[9E+09,9E+09,9E+09,9E+09,9E+09,9E+09]];
    CONST robtarget PT2a:=[[-30.267842194,-446.180487722,158.570658801],[0.000561468,0.929484006,-0.368861945,-0.00018313],[-2,-1,1,0],[9E+09,9E+09,9E+09,9E+09,9E+09,9E+09]];
    CONST robtarget PTorre2A:=[[210.216761229,-412.573624021,462.091806757],[0.333153025,0.480962472,0.784859422,-0.204156436],[-1,-1,0,0],[9E+09,9E+09,9E+09,9E+09,9E+09,9E+09]];
    CONST robtarget PTorre2A1:=[[-30.26998521,-446.179986819,198.569943565],[0.000567779,0.929486903,-0.36885461,-0.000225324],[-2,-1,1,0],[9E+09,9E+09,9E+09,9E+09,9E+09,9E+09]];
    CONST robtarget AC_C2a:=[[-241.303765497,509.814567575,50.000620305],[0.013429783,-0.950423243,0.310215827,0.016776187],[1,0,-1,0],[9E+09,9E+09,9E+09,9E+09,9E+09,9E+09]];
    CONST robtarget AC_Ra1:=[[101.131665618,-554.896940598,50.000642268],[0.014879711,0.43161718,0.901800871,-0.015504596],[-1,0,-1,0],[9E+09,9E+09,9E+09,9E+09,9E+09,9E+09]];
    CONST robtarget PsalT2:=[[-290.836185546,-433.915624341,287.541207722],[0.115922683,0.582555798,-0.758841547,0.267114547],[-2,0,1,0],[9E+09,9E+09,9E+09,9E+09,9E+09,9E+09]];


    PROC main()


        sacapieza;
        Path_10;







    ENDPROC



	PROC Path_10()
        VAR robtarget pc1;
        VAR robtarget pc2;
        VAR robtarget pc3;
        VAR robtarget pc4;
        VAR robtarget pc5;
        VAR robtarget pc6;
        VAR robtarget pc7;
        VAR robtarget pc8;
        VAR robtarget pc9;
        VAR robtarget pc10;
        VAR robtarget pc11;
        VAR robtarget pc12;
        VAR robtarget pc13;
        VAR robtarget pc14;
        VAR robtarget inicio2;



        VAR robtarget pr1;
        VAR robtarget pr2;
        VAR robtarget pr3;
        VAR robtarget pr4;
        VAR robtarget pr5;
        VAR robtarget pr6;

        VAR robtarget pt1_1;
        VAR robtarget pt1_2;
        VAR robtarget pt1_3;
        VAR robtarget pt1_4;
        VAR robtarget pt1_5;
        VAR robtarget pt1_6;
        VAR robtarget pt1_7;
        VAR robtarget pt1_8;

        VAR robtarget pt2_1;
        VAR robtarget pt2_2;
        VAR robtarget pt2_3;
        VAR robtarget pt2_4;



        VAR num rectangulo;
        VAR num cilindro;

        pt1_1:=PR1_T1;
        pt1_2:=Offs(pt1_1,0,0,40);
        pt1_3:=Offs(pt1_1,-140,0,0);
        pt1_4:=Offs(pt1_3,0,0,40);
        pt1_5:=Offs(pt1_2,0,0,40);
        pt1_6:=Offs(pt1_4,0,0,40);
        pt1_7:=Offs(pt1_1,-70,0,120);
        pt1_8:=Offs(pt1_7,0,0,40);

        pt2_1:=Offs(PR1_T2s,300,0,0);
        pt2_2:=Offs(PR2_T2s,300,0,0);
        pt2_3:=Offs(PR1_T2a,300,0,0);
        pt2_4:=Offs(pt2_3,0,0,40);

        inicio2:=Offs(pt2_3,0,0,500);





        pc1:=Offs(AC_C,0,0,40);
        pc2:=Offs(pc1,0,0,40);
        pc3:=Offs(pc2,0,0,40);

        pc4:=Offs(AC_C2a,0,0,40);
        pc5:=Offs(pc4,0,0,40);
        pc6:=Offs(pc5,0,0,40);
        pc7:=Offs(pc6,0,0,40);
        pc8:=Offs(pc7,0,0,40);
        pc9:=Offs(pc8,0,0,40);
        pc10:=Offs(AC_C2,0,0,40);
        pc11:=Offs(pc10,0,0,40);
        pc12:=Offs(pc11,0,0,40);
        pc13:=Offs(pc12,0,0,40);
        pc14:=Offs(pc13,0,0,40);






        pr1:=Offs(AC_R,0,0,40);
        pr2:=Offs(pr1,0,0,40);
        pr3:=Offs(pr2,0,0,40);
        pr4:=Offs(pr3,0,0,40);
        pr5:=Offs(pr4,0,0,40);
        pr6:=Offs(pr5,0,0,40);





        IF  (SensorCinta2=1)   THEN
                    rectangulo:=1;
                    cilindro:=0;
        ELSE
                    cilindro:=1;
                    rectangulo:=0;
        ENDIF



        IF rectangulo=1 THEN
            TEST estadoR
                CASE 1:
                    MoveL Inicio,v1000,z100,MyNewTool\WObj:=wobj0;
                    MoveL PiezaRec,v1000,z100,MyNewTool\WObj:=wobj0;
                    WaitTime 1;
                    SetDO ActivaVentosa,1;
                    MoveJ Inicio,v300,z200,MyNewTool\WObj:=wobj0;
                    MoveL PR1_T1,v300,fine,MyNewTool\WObj:=wobj0;
                    SetDO ActivaVentosa,0;
                    MoveJ Inicio,v1000,z100,MyNewTool\WObj:=wobj0;
                    estadoR:=estadoR+1;

                CASE 2:
                    MoveL Inicio,v1000,z100,MyNewTool\WObj:=wobj0;
                    MoveL PiezaRec,v1000,z100,MyNewTool\WObj:=wobj0;
                    WaitTime 1;
                    SetDO ActivaVentosa,1;
                    MoveJ Inicio,v300,z200,MyNewTool\WObj:=wobj0;
                    MoveL pt1_2,v300,fine,MyNewTool\WObj:=wobj0;
                    SetDO ActivaVentosa,0;
                    WaitTime 1;
                    MoveJ Inicio,v1000,z100,MyNewTool\WObj:=wobj0;
                    estadoR:=estadoR+1;

                CASE 3:
                    MoveL Inicio,v1000,z100,MyNewTool\WObj:=wobj0;
                    MoveL PiezaRec,v1000,z100,MyNewTool\WObj:=wobj0;
                    WaitTime 1;
                    SetDO ActivaVentosa,1;
                    MoveJ Inicio,v300,z200,MyNewTool\WObj:=wobj0;
                    MoveL pt1_3,v300,fine,MyNewTool\WObj:=wobj0;
                    SetDO ActivaVentosa,0;
                    WaitTime 1;
                    MoveJ Inicio,v1000,z100,MyNewTool\WObj:=wobj0;
                    estadoR:=estadoR+1;

                CASE 4:
                    MoveL Inicio,v1000,z100,MyNewTool\WObj:=wobj0;
                    MoveL PiezaRec,v1000,z100,MyNewTool\WObj:=wobj0;
                    WaitTime 1;
                    SetDO ActivaVentosa,1;
                    MoveJ Inicio,v300,z200,MyNewTool\WObj:=wobj0;
                    MoveL pt1_4,v300,fine,MyNewTool\WObj:=wobj0;
                    SetDO ActivaVentosa,0;
                    WaitTime 1;
                    MoveJ Inicio,v1000,z100,MyNewTool\WObj:=wobj0;
                    estadoR:=estadoR+1;

               CASE 5:
                    MoveL Inicio,v1000,z100,MyNewTool\WObj:=wobj0;
                    MoveL PiezaRec,v1000,z100,MyNewTool\WObj:=wobj0;
                    WaitTime 1;
                    SetDO ActivaVentosa,1;
                    MoveJ Inicio,v300,z200,MyNewTool\WObj:=wobj0;
                    MoveL pt2_1,v300,fine,MyNewTool\WObj:=wobj0;
                    SetDO ActivaVentosa,0;
                    WaitTime 1;
                    MoveJ Inicio,v1000,z100,MyNewTool\WObj:=wobj0;
                    estadoR:=estadoR+1;

             CASE 6:
                    MoveL Inicio,v1000,z100,MyNewTool\WObj:=wobj0;
                    MoveL PiezaRec,v1000,z100,MyNewTool\WObj:=wobj0;
                    WaitTime 1;
                    SetDO ActivaVentosa,1;
                    MoveJ Inicio,v300,z200,MyNewTool\WObj:=wobj0;
                    MoveJ inicio2,v300,fine,MyNewTool\WObj:=wobj0;
                    MoveL pt2_2,v300,fine,MyNewTool\WObj:=wobj0;
                    SetDO ActivaVentosa,0;
                    WaitTime 1;
                    MoveJ PsalT2,v300,z100,MyNewTool\WObj:=wobj0;
                    MoveJ Inicio,v1000,z100,MyNewTool\WObj:=wobj0;
                    estadoR:=estadoR+1;

           CASE 7:
                    MoveL Inicio,v1000,z100,MyNewTool\WObj:=wobj0;
                    MoveL PiezaRec,v1000,z100,MyNewTool\WObj:=wobj0;
                    WaitTime 1;
                    SetDO ActivaVentosa,1;
                    MoveJ Inicio,v300,z200,MyNewTool\WObj:=wobj0;
                    MoveJ inicio2,v300,z200,MyNewTool\WObj:=wobj0;
                    MoveJ PTorre2A,v300,z100,MyNewTool\WObj:=wobj0;
                    MoveL PT2a,v300,fine,MyNewTool\WObj:=wobj0;
                    SetDO ActivaVentosa,0;
                    WaitTime 1;
                    MoveJ Inicio,v1000,z100,MyNewTool\WObj:=wobj0;
                    estadoR:=estadoR+1;

           CASE 8:
                    MoveL Inicio,v1000,z100,MyNewTool\WObj:=wobj0;
                    MoveL PiezaRec,v1000,z100,MyNewTool\WObj:=wobj0;
                    WaitTime 1;
                    SetDO ActivaVentosa,1;
                    MoveJ Inicio,v300,z200,MyNewTool\WObj:=wobj0;
                    MoveL AC_Ra1,v300,fine,MyNewTool\WObj:=wobj0;
                    SetDO ActivaVentosa,0;
                    WaitTime 1;
                    MoveJ Inicio,v1000,z100,MyNewTool\WObj:=wobj0;
                    estadoR:=estadoR+1;



            ENDTEST
        ENDIF



        IF cilindro=1 THEN
            TEST estadoC
                CASE 1:
                    MoveL Inicio,v1000,z100,MyNewTool\WObj:=wobj0;
                    MoveL PiezaCil,v300,fine,MyNewTool\WObj:=wobj0;
                    WaitTime 1;
                    SetDO ActivaVentosa,1;
                    MoveJ Inicio,v300,z200,MyNewTool\WObj:=wobj0;
                    MoveL AC_C,v300,fine,MyNewTool\WObj:=wobj0;
                    SetDO ActivaVentosa,0;
                    WaitTime 1;
                    MoveJ Inicio,v1000,z100,MyNewTool\WObj:=wobj0;
                    estadoC:=estadoC+1;

                CASE 2:
                    MoveL Inicio,v1000,z100,MyNewTool\WObj:=wobj0;
                    MoveL PiezaCil,v300,fine,MyNewTool\WObj:=wobj0;
                    WaitTime 1;
                    SetDO ActivaVentosa,1;
                    MoveJ Inicio,v300,z200,MyNewTool\WObj:=wobj0;
                    MoveL pc1,v300,fine,MyNewTool\WObj:=wobj0;
                    SetDO ActivaVentosa,0;
                    WaitTime 1;
                    MoveJ Inicio,v1000,z100,MyNewTool\WObj:=wobj0;
                    estadoC:=estadoC+1;

                CASE 3:
                    MoveL Inicio,v1000,z100,MyNewTool\WObj:=wobj0;
                    MoveL PiezaCil,v300,fine,MyNewTool\WObj:=wobj0;
                    WaitTime 1;
                    SetDO ActivaVentosa,1;
                    MoveJ Inicio,v300,z20,MyNewTool\WObj:=wobj0;
                    MoveL pc2,v300,fine,MyNewTool\WObj:=wobj0;
                    SetDO ActivaVentosa,0;
                    WaitTime 1;
                    MoveJ Inicio,v1000,z100,MyNewTool\WObj:=wobj0;
                    estadoC:=estadoC+1;

                CASE 4:
                    MoveL Inicio,v1000,z100,MyNewTool\WObj:=wobj0;
                    MoveL PiezaCil,v300,fine,MyNewTool\WObj:=wobj0;
                    WaitTime 1;
                    SetDO ActivaVentosa,1;
                    MoveJ Inicio,v300,z200,MyNewTool\WObj:=wobj0;
                    MoveL pc3,v300,fine,MyNewTool\WObj:=wobj0;
                    SetDO ActivaVentosa,0;
                    WaitTime 1;
                    MoveJ Inicio,v1000,z100,MyNewTool\WObj:=wobj0;
                    estadoC:=estadoC+1;

                 CASE 5:
                    MoveL Inicio,v1000,z100,MyNewTool\WObj:=wobj0;
                    MoveL PiezaCil,v300,fine,MyNewTool\WObj:=wobj0;
                    WaitTime 1;
                    SetDO ActivaVentosa,1;
                    MoveJ Inicio,v1000,z200,MyNewTool\WObj:=wobj0;
                    MoveL pc4,v300,z200,MyNewTool\WObj:=wobj0;
                    SetDO ActivaVentosa,0;
                    WaitTime 1;
                    MoveJ Inicio,v1000,z100,MyNewTool\WObj:=wobj0;
                    estadoC:=estadoC+1;

                 CASE 6:
                    MoveL Inicio,v1000,z100,MyNewTool\WObj:=wobj0;
                    MoveL PiezaCil,v300,fine,MyNewTool\WObj:=wobj0;
                    WaitTime 1;
                    SetDO ActivaVentosa,1;
                    MoveJ Inicio,v300,fine,MyNewTool\WObj:=wobj0;
                    MoveL pc5,v300,fine,MyNewTool\WObj:=wobj0;
                    SetDO ActivaVentosa,0;
                    WaitTime 1;
                    MoveJ Inicio,v1000,z100,MyNewTool\WObj:=wobj0;
                    estadoC:=estadoC+1;

                  CASE 7:
                    MoveL Inicio,v1000,z100,MyNewTool\WObj:=wobj0;
                    MoveL PiezaCil,v300,fine,MyNewTool\WObj:=wobj0;
                    WaitTime 1;
                    SetDO ActivaVentosa,1;
                    MoveJ Inicio,v300,z200,MyNewTool\WObj:=wobj0;
                    MoveL pc6,v300,fine,MyNewTool\WObj:=wobj0;
                    SetDO ActivaVentosa,0;
                    WaitTime 1;
                    MoveJ Inicio,v1000,z100,MyNewTool\WObj:=wobj0;
                    estadoC:=estadoC+1;

                   CASE 8:
                    MoveL Inicio,v1000,z100,MyNewTool\WObj:=wobj0;
                    MoveL PiezaCil,v300,fine,MyNewTool\WObj:=wobj0;
                    WaitTime 1;
                    SetDO ActivaVentosa,1;
                    MoveJ Inicio,v300,z200,MyNewTool\WObj:=wobj0;
                    MoveL pc7,v300,fine,MyNewTool\WObj:=wobj0;
                    SetDO ActivaVentosa,0;
                    WaitTime 1;
                    MoveJ Inicio,v1000,z100,MyNewTool\WObj:=wobj0;
                    estadoC:=estadoC+1;

                   CASE 9:
                    MoveL Inicio,v1000,z100,MyNewTool\WObj:=wobj0;
                    MoveL PiezaCil,v300,fine,MyNewTool\WObj:=wobj0;
                    WaitTime 1;
                    SetDO ActivaVentosa,1;
                    MoveJ Inicio,v300,z200,MyNewTool\WObj:=wobj0;
                    MoveL pc8,v300,fine,MyNewTool\WObj:=wobj0;
                    SetDO ActivaVentosa,0;
                    WaitTime 1;
                    MoveJ Inicio,v1000,z100,MyNewTool\WObj:=wobj0;
                    estadoC:=estadoC+1;

                    CASE 10:
                    MoveL Inicio,v1000,z100,MyNewTool\WObj:=wobj0;
                    MoveL PiezaCil,v300,fine,MyNewTool\WObj:=wobj0;
                    WaitTime 1;
                    SetDO ActivaVentosa,1;
                    MoveJ Inicio,v300,z200,MyNewTool\WObj:=wobj0;
                    MoveL pc9,v300,fine,MyNewTool\WObj:=wobj0;
                    SetDO ActivaVentosa,0;
                    WaitTime 1;
                    MoveJ Inicio,v1000,z100,MyNewTool\WObj:=wobj0;
                    estadoC:=estadoC+1;


                    CASE 11:
                    MoveL Inicio,v1000,z100,MyNewTool\WObj:=wobj0;
                    MoveL PiezaCil,v300,fine,MyNewTool\WObj:=wobj0;
                    WaitTime 1;
                    SetDO ActivaVentosa,1;
                    MoveJ Inicio,v300,z200,MyNewTool\WObj:=wobj0;
                    MoveL pc10,v300,fine,MyNewTool\WObj:=wobj0;
                    SetDO ActivaVentosa,0;
                    WaitTime 1;
                    MoveJ Inicio,v1000,z100,MyNewTool\WObj:=wobj0;
                    estadoC:=estadoC+1;

                   CASE 12:
                    MoveL Inicio,v1000,z100,MyNewTool\WObj:=wobj0;
                    MoveL PiezaCil,v300,fine,MyNewTool\WObj:=wobj0;
                    WaitTime 1;
                    SetDO ActivaVentosa,1;
                    MoveJ Inicio,v300,z200,MyNewTool\WObj:=wobj0;
                    MoveL pc11,v300,fine,MyNewTool\WObj:=wobj0;
                    SetDO ActivaVentosa,0;
                    WaitTime 1;
                    MoveJ Inicio,v1000,z100,MyNewTool\WObj:=wobj0;
                    estadoC:=estadoC+1;

                    CASE 13:
                    MoveL Inicio,v1000,z100,MyNewTool\WObj:=wobj0;
                    MoveL PiezaCil,v300,fine,MyNewTool\WObj:=wobj0;
                    WaitTime 1;
                    SetDO ActivaVentosa,1;
                    MoveJ Inicio,v300,fine,MyNewTool\WObj:=wobj0;
                    MoveL pc12,v300,fine,MyNewTool\WObj:=wobj0;
                    SetDO ActivaVentosa,0;
                    WaitTime 1;
                    MoveJ Inicio,v1000,z100,MyNewTool\WObj:=wobj0;
                    estadoC:=estadoC+1;

                    CASE 14:
                    MoveL Inicio,v1000,z100,MyNewTool\WObj:=wobj0;
                    MoveL PiezaCil,v300,fine,MyNewTool\WObj:=wobj0;
                    WaitTime 1;
                    SetDO ActivaVentosa,1;
                    MoveJ Inicio,v300,z200,MyNewTool\WObj:=wobj0;
                    MoveL pc13,v300,fine,MyNewTool\WObj:=wobj0;
                    SetDO ActivaVentosa,0;
                    WaitTime 1;
                    MoveJ Inicio,v1000,z100,MyNewTool\WObj:=wobj0;
                    estadoC:=estadoC+1;


                    CASE 14:
                    MoveL Inicio,v1000,z100,MyNewTool\WObj:=wobj0;
                    MoveL PiezaCil,v300,fine,MyNewTool\WObj:=wobj0;
                    WaitTime 1;
                    SetDO ActivaVentosa,1;
                    MoveJ Inicio,v300,z200,MyNewTool\WObj:=wobj0;
                    MoveL pc13,v300,fine,MyNewTool\WObj:=wobj0;
                    SetDO ActivaVentosa,0;
                    WaitTime 1;
                    MoveJ Inicio,v1000,z100,MyNewTool\WObj:=wobj0;
                    estadoC:=estadoC+1;




            ENDTEST

        ENDIF






        IF estadoR>7 AND estadoC>4 THEN

            TEST estadoF
                CASE 1:
                    MoveL Inicio,v1000,z100,MyNewTool\WObj:=wobj0;
                    MoveL pc3,v300,fine,MyNewTool\WObj:=wobj0;
                    WaitTime 1;
                    SetDO ActivaVentosa,1;
                    MoveJ Inicio,v300,z200,MyNewTool\WObj:=wobj0;
                    MoveL pt1_5,v300,fine,MyNewTool\WObj:=wobj0;
                    SetDO ActivaVentosa,0;
                    WaitTime 1;
                    MoveJ Inicio,v1000,z100,MyNewTool\WObj:=wobj0;
                    estadoF:=estadoF+1;



                CASE 2:

                    MoveL pc2,v300,fine,MyNewTool\WObj:=wobj0;
                    WaitTime 1;
                    SetDO ActivaVentosa,1;
                    MoveJ Inicio,v300,z200,MyNewTool\WObj:=wobj0;
                    MoveL pt1_6,v300,fine,MyNewTool\WObj:=wobj0;
                    SetDO ActivaVentosa,0;
                    WaitTime 1;
                    MoveJ Inicio,v1000,z100,MyNewTool\WObj:=wobj0;
                    estadoF:=estadoF+1;

                CASE 3:
                    MoveL pc1,v300,fine,MyNewTool\WObj:=wobj0;
                    WaitTime 1;
                    SetDO ActivaVentosa,1;
                    MoveJ Inicio,v300,z200,MyNewTool\WObj:=wobj0;
                    MoveL PTorre2A1,v300,fine,MyNewTool\WObj:=wobj0;
                    SetDO ActivaVentosa,0;
                    WaitTime 1;
                    MoveJ Inicio,v1000,z100,MyNewTool\WObj:=wobj0;
                    estadoF:=estadoF+1;

                CASE 4:
                    MoveL AC_Ra1,v300,fine,MyNewTool\WObj:=wobj0;
                    WaitTime 1;
                    SetDO ActivaVentosa,1;
                    MoveJ Inicio,v300,z200,MyNewTool\WObj:=wobj0;
                    MoveL pt1_7,v300,fine,MyNewTool\WObj:=wobj0;
                    SetDO ActivaVentosa,0;
                    WaitTime 1;
                    MoveJ Inicio,v1000,z100,MyNewTool\WObj:=wobj0;
                    estadoF:=estadoF+1;

                CASE 5:
                    MoveL AC_C,v300,fine,MyNewTool\WObj:=wobj0;
                    WaitTime 1;
                    SetDO ActivaVentosa,1;
                    MoveJ Inicio,v300,z200,MyNewTool\WObj:=wobj0;
                    MoveL pt1_8,v300,fine,MyNewTool\WObj:=wobj0;
                    SetDO ActivaVentosa,0;
                    WaitTime 1;
                    MoveJ Inicio,v1000,z100,MyNewTool\WObj:=wobj0;
                    estadoF:=estadoF+1;
            ENDTEST


        ENDIF





	ENDPROC




    PROC sacapieza()
        SetDO ActivaSensores,0;
        SetDO ActivaSensores,1;
        SetDO Pieza,1;
        SetDO Pieza,0;
        SetDO MotorCinta,1;
        SetDO Pieza,0;
        WaitDI SensorCinta1,1;
        SetDO MotorCinta,0;
        SetDO ActivaSensores,0;
    ENDPROC

ENDMODULE

--- Backups/IRB_120_3kg_0.58m_1/RAPID/TASK1/SYSMOD/LINKEDM.sys ---
%%%
  VERSION:1
  LANGUAGE:ENGLISH
%%%

MODULE LINKEDM (SYSMODULE)

! FOLLOWER
!     Name of electronically linked follower axis used by operator at teach pendent.
      PERS string l_f_axis_name{5}       :=  ["",  "", "", "", ""];

!     Name of the mechanical unit for follower axis.
      PERS string l_f_mecunt_n{5}  :=  ["", "", "", "", ""];

!     Linked follower axis number in the mechanical unit (first axis in mech. unit is number 1).
      PERS num l_f_axis_no{5}      :=  [0,          0,   0,  0,  0];

! MASTER
!     Name of the mechanical unit for linked master axis.
      PERS string l_m_mecunt_n{5} :=  ["", "", "", "", ""];

!     Linked master axis number in the mechanical unit (first axis in mech. unit is number 1).
!     See axis number table in documentation for different master mechanical units.
      PERS num l_m_axis_no{5}     :=  [0,  0,  0,  0,  0];

! POSITION OFFSET
!     The increase of the allowed offset position between the master and follower
!     positions, used when starting AUTO mode. As soon as the offset is decreased
!     the old configurated parameter is used.
!     Example: 3 => the configurated value of allowed offset is increased 3 times.
      PERS num offset_ratio{5}       :=  [10,  10,   10,  10,  10];

! SPEED RATIO
!     Speed_ratio used in AUTO and JOG modes [ very_slow   slow    normal    fast]
!     Value 1 = max allowed manual speed.
      CONST num speed_ratio {20}      := [0.01, 0.01, 0.01, 0.01, 0.01,
                                          0.05, 0.05, 0.05, 0.05, 0.05,
                                          0.20, 0.20, 0.20, 0.20, 0.20,
                                          1.00, 1.00, 1.00, 1.00, 1.00];

! STEP SIZE
!     Displacement position used in JOG mode for each activation of positive or
!     negative movement.                  [very_short    short   normal   long]
!     Unit degees or meter.
      CONST num displacement {20}     := [0.001, 0.001, 0.001, 0.001, 0.001,
                                          0.005, 0.005, 0.005, 0.005, 0.005,
                                          0.020, 0.020, 0.020, 0.020, 0.020,
                                          0.100, 0.100, 0.100, 0.100, 0.100];


!-------------------------------------------------------------
 PROC Linked_m ()
      Linked_m_exe ;
 ENDPROC
ENDMODULE

--- Backups/IRB_120_3kg_0.58m_1/SYSPAR/EIO.cfg ---
EIO:CFG_1.0:6:1::
#
INDUSTRIAL_NETWORK:

      -Name "DeviceNet" -Label "DeviceNet Master/Slave Network" -Address "2"\
      -Simulated
#
DEVICENET_DEVICE:

      -Name "ModuloES" -Simulated
#
DEVICENET_INTERNAL_DEVICE:

      -Name "DN_Internal_Device" -VendorName "ABB Robotics"\
      -ProductName "DeviceNet Internal Slave Device"
#
EIO_SIGNAL:

      -Name "Vacuostato" -SignalType "DI" -Device "ModuloES" -Label "Vacuostado"\
      -DeviceMap "0" -Access "All"

      -Name "SensorCinta1" -SignalType "DI" -Device "ModuloES"\
      -Label "SensorCinta1" -DeviceMap "1" -Access "All"

      -Name "SensorCinta2" -SignalType "DI" -Device "ModuloES"\
      -Label "SensorCinta2" -DeviceMap "2" -Access "All"

      -Name "ActivaVentosa" -SignalType "DO" -Device "ModuloES"\
      -Label "ActivaVentosa" -DeviceMap "0" -Access "All"

      -Name "Pieza" -SignalType "DO" -Device "ModuloES" -Label "Pieza"\
      -DeviceMap "1" -Access "All"

      -Name "MotorCinta" -SignalType "DO" -Device "ModuloES" -Label "MotorCinta"\
      -DeviceMap "2" -Access "All"

      -Name "ActivaSensores" -SignalType "DO" -Device "ModuloES"\
      -Label "ActivaSensores" -DeviceMap "3" -Access "All"
